TYPE ST_MoverStatus :
STRUCT
	MoverInShortcut		: BOOL;
END_STRUCT
END_TYPE

(* stored: Version 1.1.0.1
   DUT ST_MoverStatus: Id {394eb97c-7f7c-016f-2b01-0deee4be5513} *)
